INTERFACE ITcoSequencer EXTENDS ITCoState

(*~
	<docu>
		<summary>
			Finishes the currently executed step and initiates to start the step with StepId equals to the value of the <c>inRequestedStepID</c>.
			In case that the order of the requested step is higher than the order of the currently finished step (the requested step is "after" the current one)
			the requested step is started in the same PLC cycle.
			In case that the order of the requested step is lower than the order of the currently finished step (the requested step is "before" the current one)
			the requested step is started in the next PLC cycle.
			If the requested step is not found even in the next PLC cycle, the sequencer returns the error <c>StepWithRequestedIdDoesNotExists</c>.
			<para>
				See <see cref="eSequencerError"/> for detailed description.
			</para>
		</summary>
	</docu>
~*)
METHOD RequestStep : ITcoSequencer
VAR_INPUT
	(*~
		<docu>
			<summary>
				StepId of the step to be executed.
			</summary>
		</docu>
	~*)
		inRequestedStepID : UINT;
END_VAR
END_METHOD

(*~
	<docu>
		<summary>
			This method triggers StepBackward task, that decrement current step (variable: <see cref="TcoSequencer.PlcTcoSequencer._theOrderOfTheCurrentlyExecutedStep"/> ), in case the sequencer is in step mode, and the current step is greather than zero.
		</summary>			
	</docu>	
~*)
METHOD StepBackward
END_METHOD

(*~
	<docu>
		<summary>
			Complete the actually running step, in the case the inCondition is met.
			Method is typically called inside the step as the transition method.
		</summary>			
	</docu>	
~*)
METHOD PUBLIC FINAL StepCompleteWhen : ITcoSequencer
VAR_INPUT
(*~
	<docu>
		<summary>
			The condition under which the step is completed.
		</summary>			
	</docu>	
~*)
	inCondition : BOOL;
END_VAR
END_METHOD

(*~
	<docu>
		<summary>
			This method triggers StepForward task, that increment current step (variable: <see cref="TcoSequencer.PlcTcoSequencer._theOrderOfTheCurrentlyExecutedStep"/> ), 
			in case the sequencer is in step mode, and the current step is lower than number of steps in th sequence (variable: <see cref="TcoSequencer.PlcTcoSequencer._numberOfStepsInSequence"/> ).
		</summary>			
	</docu>	
~*)
METHOD StepForward
END_METHOD

(*~
	<docu>
		<summary>
			This method triggers StepIn task, that changes the current step status from ReadyToRun to Running. 
			This causes starting the execution of the body of the current step.
		</summary>			
	</docu>	
~*)
METHOD StepIn
END_METHOD

END_INTERFACE

(* stored: Version 1.1.0.1, ProductVersion 3.1.4024.6
   Itf ITcoSequencer: Id {a8c5aaea-ce66-4699-94d6-6fc2b0db7583}
   Method RequestStep: Id {a244bce3-185f-46eb-9036-dc127d26bd08}
   Method StepBackward: Id {681ee00d-31c9-4717-8a4f-6c756dfb644e}
   Method StepCompleteWhen: Id {87266e09-a85e-45fc-bcc5-e3bf32501bbd}
   Method StepForward: Id {e42d91dc-e4a6-4639-a3ad-03d2d977e251}
   Method StepIn: Id {a6cd8de1-6571-4c77-9297-440aa85f6f9a} *)
